{attribute 'pack_mode' := '2'}
TYPE ST_NCI_CTRL :
STRUCT
  eCmd          : E_NCI_CTRL := E_NCI_CTRL.INIT;
  rOverride     : REAL := 47.11;

  sProgramName  : STRING(255);
END_STRUCT
END_TYPE

(* stored: Version 1.1.0.1, ProductVersion 3.1.4026.13
   DUT ST_NCI_CTRL: Id {409f0024-413b-084a-0caa-73fd90ffc9ad} *)
